// TIA Portal V16 export
// export: Created 2024-12-03T15:41:42.8611855Z, ExportSetting WithDefaults, DisplayName Totally Integrated Automation Portal, DisplayVersion V16 Update 6, DisplayName TIA Portal Version Control Interface, DisplayVersion V16 Update 2, DisplayName TIA Portal Openness, DisplayVersion V16 Update 6, DisplayName TIA Portal Teamcenter Gateway, DisplayVersion V16, DisplayName SINAMICS Startdrive Advanced, DisplayVersion V16 Update 5, DisplayName SINAMICS Startdrive G130, G150, S120, S150, SINAMICS MV, S210, DisplayVersion V16 Update 5, DisplayName SINAMICS Startdrive G110M, G120, G120C, G120D, G120P, G115D, DisplayVersion V16 Update 5, DisplayName STEP 7 Professional, DisplayVersion V16 Update 6, DisplayName STEP 7 Safety, DisplayVersion V16, DisplayName WinCC Advanced / Unified PC, DisplayVersion V16 Update 6
FUNCTION_BLOCK "Nord_DriveController"   // FB93, SCL
{ S7_Optimized_Access := 'FALSE' }
VERSION : 0.1
// stored: AutoNumber true, IsIECCheckEnabled false, SetENOAutomatically false, UDAEnableTagReadback false
   VAR_INPUT
      I_MotorData : "Nord_Drive_SK5xx_In_Data_UDT";
      I_Interlock : Bool;
      I_RunOverride : Bool;
      I_OverrideDirection : Bool;
      I_TimeNotRunning : Time := t#10s;
      I_TimeNotStopping : Time := t#10s;
      I_SlowStopMode : Bool;
      I_useExternalReset : Bool := TRUE;
   END_VAR
   VAR_IN_OUT
      IO_MotorStatus : "Nord_Drive_UDT";
      IO_MotorData : "Nord_Drive_SK5xx_Out_Data_UDT";
   END_VAR
   VAR DB_SPECIFIC
      S_TimeNotRunning { S7_SetPoint := 'True'} : TON_TIME;
      S_TimeNotStopping { S7_SetPoint := 'True'} : TON_TIME;
      S_TimeRunningFeedBack { S7_SetPoint := 'True'} : TON_TIME;
      S_Reset { S7_SetPoint := 'True'} : TOF_TIME;
      s_CannotStartDelay { S7_SetPoint := 'True'} : TON_TIME;
      S_SlowStopLeft { S7_SetPoint := 'True'} : TOF_TIME;
      S_SlowStopRight { S7_SetPoint := 'True'} : TOF_TIME;
      CannotStartErrorDelay : TON_TIME;
      S_SpeedSetPoint : Int;
   END_VAR
   VAR
      cycleCounter : "CycleRun";
      AlarmNotRunning : Program_Alarm;
      AlarmNotStopping : Program_Alarm;
      AlarmErrorActive : Program_Alarm;
      AlarmCannotStart : Program_Alarm;
      AlarmNotConnected : Program_Alarm;
      AlarmEmergencyStopActive : Program_Alarm;
      AlarmWarningActive : Program_Alarm;
      WarningManualOverrideActive { S7_SetPoint := 'True'} : Program_Alarm;
   END_VAR
   VAR DB_SPECIFIC
      T_ZoneInfo { ExternalAccessible := 'False'; ExternalVisible := 'False'; ExternalWritable := 'False'} : "ZoneInfo";
      T_Appstate { ExternalAccessible := 'False'; ExternalVisible := 'False'; ExternalWritable := 'False'} : "ApplicationState_UDT";
      Alarm { S7_SetPoint := 'True'} : "AlarmInfo_UDT";
   END_VAR
   VAR_TEMP
      T_dummy : UInt;
      T_Direction : Bool;
      T_RunLeftCmd : Bool;
      T_RunRightCmd : Bool;
      T_EnableOperation : Bool;
      T_SlowStopSetting : Time;
   END_VAR
BEGIN
   #T_ZoneInfo := "ApplicationState_DB".ZoneNames[#IO_MotorStatus.Zone];
   #T_Appstate := "ApplicationState_DB".Appstate[#T_ZoneInfo.AppStateIndex];
   #T_RunLeftCmd := FALSE;
   #T_RunRightCmd := FALSE;

   IF "RunTime_DB".CycleRun = #T_ZoneInfo.AppStateIndex THEN
       #cycleCounter(I_Start := 1,
                     I_End := 7);
   END_IF;

   REGION Copy commands

       #IO_MotorStatus.Status.ManualCommandsDisabled := 0;

       //Always false commands
       #IO_MotorData.xStart48011_Takt := 0;
       #IO_MotorData.xStart48012_Home := 0;
       #IO_MotorData.Parameterset_LSB := 0;
       #IO_MotorData.Parameterset_MSB := 0;

       //Alwas true commands
       #IO_MotorData.ActivatePower := 1;
       #IO_MotorData.EmergencyOk := 1;
       #IO_MotorData.EnableRampGenerator := 1;
       #IO_MotorData.EnableSetPointRampGenerator := 1;
       #IO_MotorData.xEnSetp := 1;
       #IO_MotorData.xCrtlData := 1;

       //Run motor commands
       #T_RunLeftCmd := 0;
       #T_RunRightCmd := 0;
       #T_EnableOperation := 0;
       #IO_MotorData.CmdLeftDirection := 0;
       #IO_MotorData.CmdRightDirection := 0;
       #IO_MotorData.EnableOperation := 0;

       //Save ccommands
       #IO_MotorData.CmdReadyForOPeration := 0;
       #IO_MotorData.ActivatePower := 1;

       //Auto mode
       IF #T_Appstate.States.AutoModeActivated.State AND NOT #IO_MotorStatus.Status.ManualModeActive
           AND #IO_MotorStatus.Alarms.AlarmStatus = 0 THEN
           #T_RunLeftCmd := #IO_MotorStatus.Cmd.DirectionAuto AND #IO_MotorStatus.Cmd.OnAuto;
           #T_RunRightCmd := NOT #IO_MotorStatus.Cmd.DirectionAuto AND #IO_MotorStatus.Cmd.OnAuto;
           #S_SpeedSetPoint := REAL_TO_INT(#IO_MotorStatus.Cmd.SpeedAuto);
       END_IF;

       //Manual mode
       IF  #IO_MotorStatus.Status.ManualModeActive  THEN

           IF NOT #IO_MotorStatus.Settings.AllowManualDirection THEN
               #T_Direction := #IO_MotorStatus.Settings.DefaultDirection;
           ELSE
               #T_Direction := #IO_MotorStatus.Cmd.DirectionManual;
           END_IF;

           #T_RunLeftCmd := #T_Direction AND #IO_MotorStatus.Cmd.OnManual;
           #T_RunRightCmd := NOT #T_Direction AND #IO_MotorStatus.Cmd.OnManual;
           #S_SpeedSetPoint := REAL_TO_INT(#IO_MotorStatus.Cmd.SpeedManual);
       END_IF;

       //Turn commands of if manual mode is deactivated
       IF NOT #IO_MotorStatus.Status.ManualModeActive  THEN
           #IO_MotorStatus.Cmd.OnManual := 0;
           #IO_MotorStatus.Cmd.DirectionManual := 0;
           #IO_MotorStatus.Status.ManualCommandsDisabled := 1;
       END_IF;


       REGION Slow stop MODe
           IF #I_SlowStopMode AND ABS_INT(IN:= #IO_MotorStatus.Status.ActualSpeed) > 10 THEN
               #T_SlowStopSetting := t#500ms;
           ELSE
               #T_SlowStopSetting := t#0ms;
           END_IF;

           #S_SlowStopLeft(IN := #T_RunLeftCmd AND NOT #IO_MotorData.CmdRightDirection AND NOT #IO_MotorStatus.Cmd.Interlock,
                               PT := #T_SlowStopSetting,
                               Q=>#IO_MotorData.CmdLeftDirection);


               #S_SlowStopRight(IN := #T_RunRightCmd AND NOT #IO_MotorData.CmdLeftDirection AND NOT #IO_MotorStatus.Cmd.Interlock,
                                PT := #T_SlowStopSetting,
                                Q => #IO_MotorData.CmdRightDirection);

               //Set slow speed when there is no run command
               IF NOT #T_RunLeftCmd AND NOT #T_RunRightCmd THEN
                   #IO_MotorData.MotorSetpointSpeed := REAL_TO_INT(IN:=10.0) * (16384 / 100);
               ELSE
                   #IO_MotorData.MotorSetpointSpeed := (REAL_TO_INT(IN:=#S_SpeedSetPoint) * (16384 / 100));
               END_IF;

               #IO_MotorData.EnableOperation := #IO_MotorData.CmdLeftDirection OR #IO_MotorData.CmdRightDirection;
               #IO_MotorData.CmdReadyForOPeration := #IO_MotorData.EnableOperation;

       END_REGION

       IF #I_RunOverride THEN
           #IO_MotorData.CmdLeftDirection := #I_OverrideDirection;
           #IO_MotorData.CmdRightDirection := NOT #I_OverrideDirection;
           #IO_MotorData.EnableOperation := #IO_MotorData.CmdLeftDirection OR #IO_MotorData.CmdRightDirection;
           #IO_MotorData.CmdReadyForOPeration := #IO_MotorData.EnableOperation;
       END_IF;

   END_REGION

   REGION BUILD NAME

       IF NOT #Alarm.init OR #IO_MotorStatus.info.Name = '' OR "HMI_DB".ReloadSettings.signal THEN
           #IO_MotorStatus.info.Name := "buildObjectName"(I_Symbolname := GetSymbolName(variable := #IO_MotorStatus, size := 100));
           #Alarm.info := "buildAlarmInfo"(I_ObjectName := #IO_MotorStatus.info.Name, I_ZoneIndex := #IO_MotorStatus.Zone, I_ZoneName := #T_ZoneInfo.ZoneName);
           #Alarm.init := true;
       END_IF;

   END_REGION

   REGION alarms

       REGION Time NOT running

           #S_TimeNotRunning(IN := #IO_MotorData.EnableOperation
                             AND NOT #IO_MotorStatus.Alarms.NotOnTImedOut.Active AND #IO_MotorStatus.Status.ActualSpeed = 0,
                             PT := t#10s);

           IF #S_TimeNotRunning.Q THEN
               #IO_MotorStatus.Alarms.NotOnTImedOut.Active := true;
           END_IF;


       END_REGION

       REGION Time NOT stopping

           #S_TimeNotStopping(IN := NOT #IO_MotorData.EnableOperation AND #IO_MotorStatus.Status.Running,
                              PT := t#10s);

           IF #S_TimeNotStopping.Q THEN
               #IO_MotorStatus.Alarms.NotOffTimedOut.Active := TRUE;
           END_IF;

       END_REGION

       REGION Error active

           IF #I_MotorData.ErrorActive THEN
               #IO_MotorStatus.Alarms.ErrorFromDrive.Active := true;
           END_IF;

       END_REGION

       REGION Cannot start error

           #s_CannotStartDelay(IN := #I_MotorData.CannotStartError AND #IO_MotorData.EnableOperation,
                               PT := t#1s);

           IF #s_CannotStartDelay.Q THEN
               #IO_MotorStatus.Alarms.CannotStartError.Active := true;
           END_IF;

       END_REGION

       REGION Device not connected

           // IF NOT #I_MotorData.BusControllerActive AND NOT #I_MotorData.PowerOn THEN //OR NOT #I_MotorData.ReadyToStart THEN
           //     #IO_MotorStatus.Alarms.Disconnected.Active := true;
           // END_IF;

           #IO_MotorStatus.Alarms.Disconnected.Active := NOT #I_MotorData.BusControllerActive AND NOT #I_MotorData.PowerOn;

       END_REGION

       REGION Emergency stop active

           #IO_MotorStatus.Alarms.EmergencyStopActive.Active := #I_MotorData.EmergencyStoPActive;
           #IO_MotorStatus.Alarms.EmergencyStopActive.Active := 0;

       END_REGION

       REGION Warning on drive active

           #IO_MotorStatus.Alarms.WarningFromDrive.Active := #I_MotorData.WarningActive;

       END_REGION

       REGION PROGRAM ALARMS

           IF #cycleCounter.O_Cycle = 1 AND "RunTime_DB".CycleRun = #T_ZoneInfo.AppStateIndex THEN

               #AlarmNotRunning(SIG := #IO_MotorStatus.Alarms.NotOnTImedOut.Active,
                                SD_1 := #Alarm.info,
                                SD_2 := #T_ZoneInfo.ZoneName,
                                SD_3 := #IO_MotorStatus.info.Name);

           END_IF;

           IF #cycleCounter.O_Cycle = 2 AND "RunTime_DB".CycleRun = #T_ZoneInfo.AppStateIndex THEN

               #AlarmNotStopping(SIG := #IO_MotorStatus.Alarms.NotOffTimedOut.Active,
                                 SD_1 := #Alarm.info,
                                 SD_2 := #T_ZoneInfo.ZoneName,
                                 SD_3 := #IO_MotorStatus.info.Name);
           END_IF;
           IF #cycleCounter.O_Cycle = 3 AND "RunTime_DB".CycleRun = #T_ZoneInfo.AppStateIndex THEN

               #AlarmErrorActive(SIG := #IO_MotorStatus.Alarms.ErrorFromDrive.Active,
                                 SD_1 := #Alarm.info,
                                 SD_2 := #T_ZoneInfo.ZoneName,
                                 SD_3 := #IO_MotorStatus.info.Name);
           END_IF;
           IF #cycleCounter.O_Cycle = 4 AND "RunTime_DB".CycleRun = #T_ZoneInfo.AppStateIndex THEN

               #AlarmCannotStart(SIG := #IO_MotorStatus.Alarms.CannotStartError.Active,
                                 SD_1 := #Alarm.info,
                                 SD_2 := #T_ZoneInfo.ZoneName,
                                 SD_3 := #IO_MotorStatus.info.Name);
           END_IF;
           IF #cycleCounter.O_Cycle = 5 AND "RunTime_DB".CycleRun = #T_ZoneInfo.AppStateIndex THEN

               #AlarmNotConnected(SIG := #IO_MotorStatus.Alarms.Disconnected.Active,
                                  SD_1 := #Alarm.info,
                                  SD_2 := #T_ZoneInfo.ZoneName,
                                  SD_3 := #IO_MotorStatus.info.Name);
           END_IF;
           IF #cycleCounter.O_Cycle = 6 AND "RunTime_DB".CycleRun = #T_ZoneInfo.AppStateIndex THEN

               #AlarmEmergencyStopActive(SIG := #IO_MotorStatus.Alarms.EmergencyStopActive.Active,
                                         SD_1 := #Alarm.info,
                                         SD_2 := #T_ZoneInfo.ZoneName,
                                         SD_3 := #IO_MotorStatus.info.Name);
           END_IF;
           IF #cycleCounter.O_Cycle = 7 AND "RunTime_DB".CycleRun = #T_ZoneInfo.AppStateIndex THEN

               #AlarmWarningActive(SIG := #IO_MotorStatus.Alarms.WarningFromDrive.Active,
                                   SD_1 := #Alarm.info,
                                   SD_2 := #T_ZoneInfo.ZoneName,
                                   SD_3 := #IO_MotorStatus.info.Name);

           END_IF;

       END_REGION

   END_REGION

   REGION Create alarm status

       #IO_MotorStatus.Alarms.AlarmStatus.%X0 := #IO_MotorStatus.Alarms.NotOnTImedOut.Active;
       #IO_MotorStatus.Alarms.AlarmStatus.%X1 := #IO_MotorStatus.Alarms.NotOffTimedOut.Active;
       #IO_MotorStatus.Alarms.AlarmStatus.%X2 := #IO_MotorStatus.Alarms.ErrorFromDrive.Active;
       #IO_MotorStatus.Alarms.AlarmStatus.%X3 := #IO_MotorStatus.Alarms.CannotStartError.Active;
       #IO_MotorStatus.Alarms.AlarmStatus.%X4 := #IO_MotorStatus.Alarms.EmergencyStopActive.Active;
       #IO_MotorStatus.Alarms.AlarmStatus.%X5 := #IO_MotorStatus.Alarms.Disconnected.Active;

       IF #IO_MotorStatus.Alarms.AlarmStatus > 0 THEN
           "ApplicationState_DB".Appstate[#T_ZoneInfo.AppStateIndex].Alarms.AlarmActiveInternalPLC := TRUE;
       END_IF;

   END_REGION

   REGION Turn commands off on error

       #IO_MotorData.EmergencyOk := #T_Appstate.States.EmergencyOk.State;
       #IO_MotorData.ActivatePower := #IO_MotorData.EmergencyOk;

       IF NOT #I_RunOverride THEN

           IF (#IO_MotorStatus.Alarms.AlarmStatus > 0)
               OR NOT #T_Appstate.States.EmergencyOk.State
               OR (#I_Interlock AND #IO_MotorStatus.Status.ManualCommandsDisabled)
           THEN
               #IO_MotorData.CmdLeftDirection := 0;
               #IO_MotorData.CmdRightDirection := 0;
               #IO_MotorData.EnableOperation := 0;
               #IO_MotorData.CmdReadyForOPeration := 0;
           END_IF;
       END_IF;

       #CannotStartErrorDelay(IN:= NOT #IO_MotorStatus.Alarms.CannotStartError.Active,
                              PT:=t#250ms);

       IF NOT #CannotStartErrorDelay.Q OR #IO_MotorStatus.Alarms.ErrorFromDrive.Active THEN
           #IO_MotorData.CmdLeftDirection := 0;
           #IO_MotorData.CmdRightDirection := 0;
           #IO_MotorData.EnableOperation := 0;
           #IO_MotorData.CmdReadyForOPeration := 0;
       END_IF;

   END_REGION

   REGION Create status

       #IO_MotorStatus.Status.ManualModeActive := #T_Appstate.States.ManualModeActivated.State;
       #IO_MotorStatus.Status.Interlocked := #I_Interlock OR #IO_MotorStatus.Cmd.Interlock;
       #IO_MotorStatus.Status.ActualDirection := #I_MotorData.MotorIsRunningLeft AND NOT #I_MotorData.MotorIsRunningRight;
       #IO_MotorStatus.Status.ActualSpeed := REAL_TO_INT(IN := ( INT_TO_REAL(IN:=#I_MotorData.ActualSpeed) * 100.0) / 16384.0);
       #IO_MotorStatus.Status.PowerOn := #I_MotorData.PowerOn;
       #IO_MotorStatus.Status.ReadyForOperaiton := #I_MotorData.ReadyForOperation;
       #IO_MotorStatus.Status.ReadyToStart := #I_MotorData.ReadyToStart;

       #IO_MotorStatus.Status.Status.%X0 := #IO_MotorStatus.Status.Interlocked;
       #IO_MotorStatus.Status.Status.%X2 := #IO_MotorStatus.Status.ManualModeActive;

       #IO_MotorStatus.Status.Status.%X4 := #IO_MotorStatus.Status.ReadyToStart;
       #IO_MotorStatus.Status.Status.%X5 := #IO_MotorStatus.Status.ReadyForOperaiton;
       #IO_MotorStatus.Status.Status.%X6 := #IO_MotorStatus.Status.PowerOn;

       #IO_MotorStatus.Status.CmdRunManualActive :=
       (#IO_MotorData.CmdLeftDirection OR #T_RunLeftCmd OR #T_RunRightCmd OR #IO_MotorData.CmdRightDirection)
       AND  #IO_MotorStatus.Status.ManualModeActive ;

   END_REGION

   REGION Reset 

       #S_Reset(IN := (#T_Appstate.Hmi_Buttons.reset.state.State AND #I_useExternalReset)
                OR #IO_MotorStatus.Cmd.Reset
                OR #I_RunOverride,
                PT := t#1s,
                Q => #IO_MotorData.ResetError);

       IF #IO_MotorData.ResetError THEN
           #IO_MotorStatus.Alarms.NotOnTImedOut.Active := 0;
           #IO_MotorStatus.Alarms.NotOffTimedOut.Active:= 0;
           #IO_MotorStatus.Alarms.ErrorFromDrive.Active:= 0;
           #IO_MotorStatus.Alarms.CannotStartError.Active := 0;
           #IO_MotorStatus.Alarms.EmergencyStopActive.Active := 0;
           #IO_MotorStatus.Alarms.Disconnected.Active := 0;
       END_IF;

   END_REGION

   REGION Running feedback

       #IO_MotorStatus.Status.Running := #I_MotorData.Running AND
       (#IO_MotorStatus.Status.ActualSpeed > 0 OR #IO_MotorStatus.Status.ActualSpeed < 0)
       AND #IO_MotorData.EnableOperation AND (#IO_MotorData.CmdLeftDirection OR #IO_MotorData.CmdRightDirection);

       #IO_MotorStatus.Status.Status.%X1 := #IO_MotorStatus.Status.Running;

   END_REGION

   REGION common status
       #IO_MotorStatus.Commonstatus := 0;
       IF #IO_MotorStatus.Status.Running THEN
           #IO_MotorStatus.Commonstatus := 1;
       END_IF;

       IF #IO_MotorStatus.Alarms.AlarmStatus > 1 AND NOT #IO_MotorStatus.Alarms.EmergencyStopActive.Active THEN
           #IO_MotorStatus.Commonstatus := 2;
       END_IF;
   END_REGION

   IF #IO_MotorStatus.Cmd.Reset THEN
       #IO_MotorStatus.Cmd.Reset := 0;
   END_IF;
END_FUNCTION_BLOCK
